FUNCTION_BLOCK MY_X2Y2_J (* Compute X^2-Y^2 in Java *)
  (* Standard: 61499-1 *)
  (* Version 0.2, 2011-08-21, JHC, Holobloc Inc, Moved algorithm text to a CDATA section. *)
  (* Version 0.1, 2006-09-06, JHC, Holobloc Inc, Made a SimpleFB. *)
  (* Version 0.0, 2001-10-09, JHC, Rockwell Automation *)
  (* Compiler header: package fb.rt.student; import fb.rt.math.*; *)
  (* Compiler classdef: SimpleFB *)
  (* Compiler Java IBM Jikes 1.0.6 *)
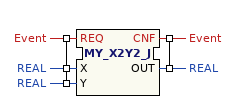
  EVENT_INPUT
    REQ WITH X, Y;
  END_EVENT
  EVENT_OUTPUT
    CNF WITH OUT;
  END_EVENT
  VAR_INPUT
    X : REAL;
    Y : REAL;
  END_VAR
  VAR_OUTPUT
    OUT : REAL;
  END_VAR
  ALGORITHM REQ IN Java:
OUT.value = (X.value-Y.value)*(X.value+Y.value);
  END_ALGORITHM
END_FUNCTION_BLOCK
